Staubli VAL3: onF7Event.pgx

program onF7Event(bool& x_bSave[] (dimensions=1))
begin
  // look if the bButton is enable
  if bButton[6]
    //
    // CHANGE THE PROFILE
    //
    call passwd(x_bSave)
  endIf
end
